{attribute 'GeneratedUsingTerminal: EPP6002-0002-0018'}
{attribute addProperty BoxType "EPP6002-0002-0018"}
{attribute addProperty Id "StatusAT %I*UINT2Data_InAT %I*ARRAY[0..21] OF USINT22"}
{attribute addProperty CRC "1367962124"}
{attribute addProperty Size "24"}
TYPE COM_TxPDO_Map_Inputs_Channel_6C2FC202 :
STRUCT
	{attribute addProperty Name "Status"}
	Status AT %I* : UINT;
	{attribute addProperty Name "Data_In"}
	Data_In AT %I* : ARRAY[0..21] OF USINT;
END_STRUCT
END_TYPE

(* stored: Version 1.2.0.0, ProductVersion 3.1.4024.9
   DUT COM_TxPDO_Map_Inputs_Channel_6C2FC202: Id {58479201-7498-457b-928b-22112abbeed7} *)
